ABB RobotStudio station: Aristides_20220202-142745.rsstn

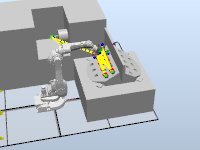
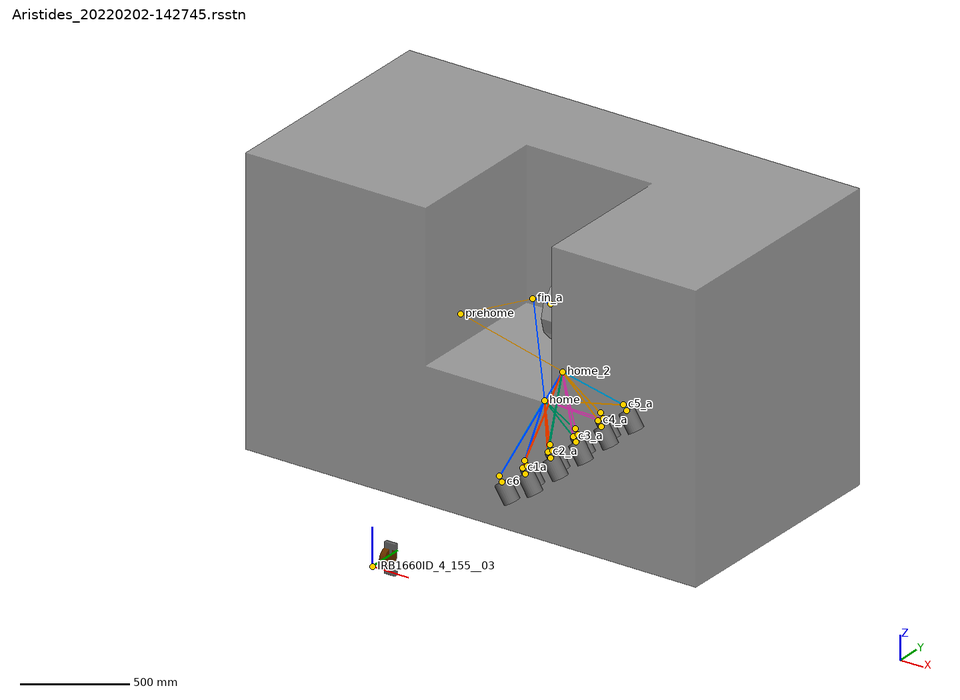
[picture v1: parts stored in the station drawn from their meshes, with robot base, taught points and paths (robot models come from the ABB library and are not in the file)]
Station Aristides (saved by RobotStudio 21.4.9700.0)
Controller Controller3
  mechanical unit ROB_1: IRB1660ID_4_155__03, 6 joints, base frame (0, 0, 0) mm
Layout (positions relative to the parent item):
  - IRB1660ID_4_155__03 [mechanism, from Robots\IRB1660ID_4_155__03.rslib] at (0, 0, 0) mm; joint values [0, 0, 0, 0, 0.5236, 0] (rad or m)
  - Pinza_1 [mechanism, from Efectores_finales - Copy\Pinza_1.rslib] at (944.87, 0, 1229) mm, rotated rx 180 ry 60 rz 180 deg; joint values [0, 0] (rad or m)
  - Torno [part] at (-1172.42, 1966.27, 0) mm, rotated rx 0 ry 0 rz 180 deg, size 2500 x 1300 x 1500 mm
  - Fence_740 [graphiccomponentgroup, from Equipment\Fence_740.rslib] at (-1160.76, -802.49, 0) mm
    - Body 1 [part, from Equipment\Fence_740.rslib]
    - Body 2 [part, from Equipment\Fence_740.rslib]
  - Fence_2500 [graphiccomponentgroup, from Equipment\Fence_2500.rslib] at (1297.15, -826.85, 0) mm, rotated rx 0 ry 0 rz 90 deg
    - Body 1 [part, from Equipment\Fence_2500.rslib]
    - Body 2 [part, from Equipment\Fence_2500.rslib]
  - Fence_740_2 [graphiccomponentgroup, from Equipment\Fence_740.rslib] at (-1148.66, -57.63, 0) mm
    - Body 1 [part, from Equipment\Fence_740.rslib]
    - Body 2 [part, from Equipment\Fence_740.rslib]
  - c5 [part] at (1213.21, 355.81, 885.53) mm, rotated rx 0 ry -32 rz 0 deg, size 80 x 79.4 x 100 mm
  - c3 [part] at (1213.21, -44.2, 885.53) mm, rotated rx 0 ry -32 rz 0 deg, size 80 x 79.4 x 100 mm
  - c2 [part] at (1213.21, -244.19, 885.53) mm, rotated rx 0 ry -32 rz 0 deg, size 80 x 79.4 x 100 mm
  - c8 [part] at (1084.59, -44.2, 808.36) mm, rotated rx 0 ry -32 rz 0 deg, size 80 x 79.4 x 100 mm
  - c4 [part] at (1213.21, 155.81, 885.53) mm, rotated rx 0 ry -32 rz 0 deg, size 80 x 79.4 x 100 mm
  - c7 [part] at (1084.59, -244.19, 808.36) mm, rotated rx 0 ry -32 rz 0 deg, size 80 x 79.4 x 100 mm
  - c6 [part] at (1084.59, -444.19, 808.36) mm, rotated rx 0 ry -32 rz 0 deg, size 80 x 79.4 x 100 mm
  - c9 [part] at (1084.59, 155.81, 808.36) mm, rotated rx 0 ry -32 rz 0 deg, size 80 x 79.4 x 100 mm
  - c10 [part] at (1084.59, 355.81, 808.36) mm, rotated rx 0 ry -32 rz 0 deg, size 80 x 79.4 x 100 mm
  - fin [part] at (377.58, 1016.27, 1000) mm, size 100 x 79.4 x 80 mm
  - c0 [part] at (277.58, 1016.27, 1000) mm, size 100 x 79.4 x 80 mm
  - Positioner [smart component, from Components\Positioner.rslib]
      properties: Object=(none); Position=[0 0 0]; Orientation=[0 0 0]; Reference=Global; ReferenceObject=(none)
  - Detacher [smart component, from Components\Detacher.rslib]
      properties: Child=(none); KeepPosition=true
  - Attacher [smart component, from Components\Attacher.rslib]
      properties: Parent=Pinza_2; Flange=0; Child=(none); Mount=false; Offset=[0 0 0]; Orientation=[0 0 0]
  - CollisionSensor [smart component, from Components\CollisionSensor.rslib]
      properties: Object1=Pinza_2; Object2=c1; NearMiss=0.01; Part1=(none); Part2=(none); CollisionType=0
  - CollisionSensor_2 [smart component, from Components\CollisionSensor.rslib]
      properties: Object1=(none); Object2=(none); NearMiss=0; Part1=(none); Part2=(none); CollisionType=0
  - c1 [part] at (1213.21, -444.19, 885.53) mm, rotated rx 0 ry -32 rz 0 deg, size 80 x 79.4 x 100 mm
  - Efector final 2 [part] at (70, 0, -80) mm, rotated rx 0 ry -90 rz -180 deg, size 100 x 99.5 x 30 mm
  - Pinza1_5 [part] at (130, 10, -10) mm, rotated rx 0 ry 0 rz 180 deg, size 60 x 20 x 60 mm
  - Pinza1_6 [part] at (130, -10, 150) mm, rotated rx 180 ry 0 rz 180 deg, size 60 x 20 x 60 mm
    - Pinza_2_1 [frame] at (30, 10, 80) mm, rotated rx 0 ry -90 rz 0 deg
  - Pinza_2 [mechanism, from Efectores_finales\PINZA2.rslib] at (944.87, 0, 1229) mm, rotated rx 180 ry 60 rz 180 deg; joint values [0, 0] (rad or m)
  - mesa_giratoria [smart component, from Efectores_finales\mesa_giratoria.rslib] at (1381.81, -44.2, 0) mm
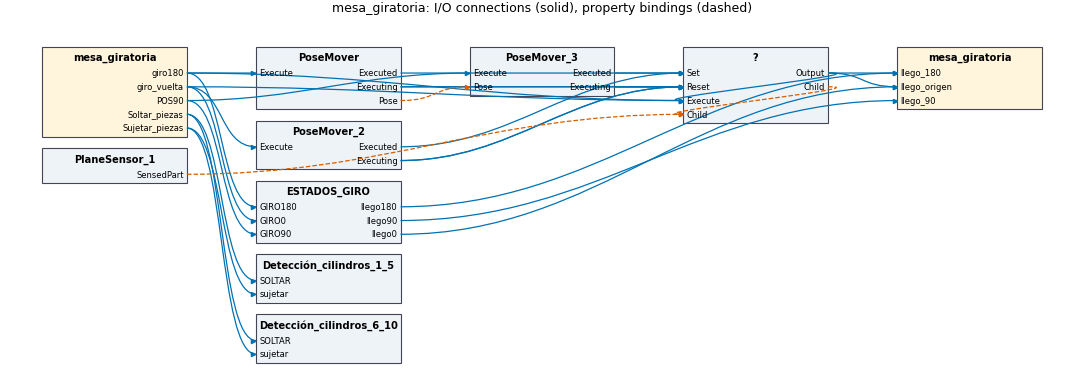
      connections:
        mesa_giratoria.giro180 -> PoseMover.Execute
        mesa_giratoria.giro_vuelta -> PoseMover_2.Execute
        PoseMover.Executed -> ?.Set
        ?.Output -> mesa_giratoria.llego_180
        PoseMover_2.Executed -> ?.Set
        ?.Output -> mesa_giratoria.llego_origen
        PoseMover_2.Executing -> ?.Reset
        PoseMover.Executing -> ?.Reset
        ?.Output -> ?.Execute
        mesa_giratoria.giro_vuelta -> ?.Execute
        mesa_giratoria.giro180 -> ?.Execute
        mesa_giratoria.POS90 -> PoseMover_3.Execute
        PoseMover_3.Executed -> ?.Set
        PoseMover.Executing -> ?.Reset
        PoseMover_2.Executing -> ?.Reset
        PoseMover_3.Executing -> ?.Reset
        PoseMover_3.Executing -> ?.Reset
        mesa_giratoria.giro180 -> ESTADOS_GIRO.GIRO180
        mesa_giratoria.giro_vuelta -> ESTADOS_GIRO.GIRO0
        mesa_giratoria.POS90 -> ESTADOS_GIRO.GIRO90
        ESTADOS_GIRO.llego180 -> mesa_giratoria.llego_180
        ESTADOS_GIRO.llego90 -> mesa_giratoria.llego_90
        ESTADOS_GIRO.llego0 -> mesa_giratoria.llego_origen
        mesa_giratoria.Soltar_piezas -> Detección_cilindros_1_5.SOLTAR
        mesa_giratoria.Soltar_piezas -> Detección_cilindros_6_10.SOLTAR
        mesa_giratoria.Sujetar_piezas -> Detección_cilindros_1_5.sujetar
        mesa_giratoria.Sujetar_piezas -> Detección_cilindros_6_10.sujetar
        PlaneSensor_1.SensedPart => ?.Child
        ?.Child => ?.Child
        PoseMover.Pose => PoseMover_3.Pose
    - Detección_cilindros_6_10 [smart component, from Efectores_finales\mesa_giratoria.rslib]
        connections:
          Detección_cilindros_6_10.SOLTAR -> Deteccion6.liberar
          Detección_cilindros_6_10.SOLTAR -> Deteccion10.liberar
          Detección_cilindros_6_10.SOLTAR -> Deteccion7.liberar
          Detección_cilindros_6_10.SOLTAR -> Deteccion8.liberar
          Detección_cilindros_6_10.SOLTAR -> Deteccion9.liberar
          Detección_cilindros_6_10.sujetar -> Deteccion6.Fijar
          Detección_cilindros_6_10.sujetar -> Deteccion10.Fijar
          Detección_cilindros_6_10.sujetar -> Deteccion7.Fijar
          Detección_cilindros_6_10.sujetar -> Deteccion9.Fijar
          Detección_cilindros_6_10.sujetar -> Deteccion8.Fijar
      - Deteccion6 [smart component, from Efectores_finales\mesa_giratoria.rslib]
        - Attacher_6 [smart component, from Components\Attacher.rslib]
            properties: Parent=Mi_mecanismo; Flange=0; Child=c6; Mount=false; Offset=[0 0 0]; Orientation=[0 0 0]
        - PlaneSensor_6 [smart component, from Components\PlaneSensor.rslib] at (-613.43, 800, 257.08) mm, rotated rx 0 ry 42 rz 0 deg
            properties: Origin=[0.0459897083517545 -0.4 1.14120505334971]; Axis1=[0.0787846202409767 0 0.0138918542133544]; Axis2=[0 0.04 0]; SensedPart=(none)
          - _sensorPart_ [part, from Efectores_finales\mesa_giratoria.rslib]
        - Detacher_6 [smart component, from Components\Detacher.rslib]
            properties: Child=(none); KeepPosition=true
      - Deteccion7 [smart component, from Efectores_finales\mesa_giratoria.rslib]
        - Attacher_7 [smart component, from Components\Attacher.rslib]
            properties: Parent=Mi_mecanismo; Flange=0; Child=c7; Mount=false; Offset=[0 0 0]; Orientation=[0 0 0]
        - PlaneSensor_7 [smart component, from Components\PlaneSensor.rslib] at (-613.43, 600, 257.08) mm, rotated rx 0 ry 42 rz 0 deg
            properties: Origin=[0.0459897083517545 -0.4 1.14120505334971]; Axis1=[0.0787846202409767 0 0.0138918542133544]; Axis2=[0 0.04 0]; SensedPart=(none)
          - _sensorPart_ [part, from Efectores_finales\mesa_giratoria.rslib]
        - Detacher_7 [smart component, from Components\Detacher.rslib]
            properties: Child=(none); KeepPosition=true
      - Deteccion8 [smart component, from Efectores_finales\mesa_giratoria.rslib]
        - Attacher_8 [smart component, from Components\Attacher.rslib]
            properties: Parent=Mi_mecanismo; Flange=0; Child=c8; Mount=false; Offset=[0 0 0]; Orientation=[0 0 0]
        - PlaneSensor_8 [smart component, from Components\PlaneSensor.rslib] at (-613.43, 400, 257.08) mm, rotated rx 0 ry 42 rz 0 deg
            properties: Origin=[0.0459897083517545 -0.4 1.14120505334971]; Axis1=[0.0787846202409767 0 0.0138918542133544]; Axis2=[0 0.04 0]; SensedPart=(none)
          - _sensorPart_ [part, from Efectores_finales\mesa_giratoria.rslib]
        - Detacher_8 [smart component, from Components\Detacher.rslib]
            properties: Child=(none); KeepPosition=true
      - Deteccion9 [smart component, from Efectores_finales\mesa_giratoria.rslib]
        - PlaneSensor_9 [smart component, from Components\PlaneSensor.rslib] at (-613.43, 0, 257.08) mm, rotated rx 0 ry 42 rz 0 deg
            properties: Origin=[0.0459897083517545 -0.4 1.14120505334971]; Axis1=[0.0787846202409767 0 0.0138918542133544]; Axis2=[0 0.04 0]; SensedPart=(none)
          - _sensorPart_ [part, from Efectores_finales\mesa_giratoria.rslib]
        - Attacher_9 [smart component, from Components\Attacher.rslib]
            properties: Parent=Mi_mecanismo; Flange=0; Child=c9; Mount=true; Offset=[0 0 0]; Orientation=[0 0 0]
        - Detacher_9 [smart component, from Components\Detacher.rslib]
            properties: Child=(none); KeepPosition=true
      - Deteccion10 [smart component, from Efectores_finales\mesa_giratoria.rslib]
        - Attacher_10 [smart component, from Components\Attacher.rslib] at (-100, -800, -200) mm
            properties: Parent=Mi_mecanismo; Flange=0; Child=c10; Mount=false; Offset=[0 0 0]; Orientation=[0 0 0]
        - PlaneSensor_10 [smart component, from Components\PlaneSensor.rslib] at (-613.43, 200, 257.08) mm, rotated rx 0 ry 42 rz 0 deg
            properties: Origin=[0.0459897083517545 -0.4 1.14120505334971]; Axis1=[0.0787846202409767 0 0.0138918542133544]; Axis2=[0 0.04 0]; SensedPart=(none)
          - _sensorPart_ [part, from Efectores_finales\mesa_giratoria.rslib]
        - Detacher_10 [smart component, from Components\Detacher.rslib]
            properties: Child=(none); KeepPosition=true
    - Detección_cilindros_1_5 [smart component, from Efectores_finales\mesa_giratoria.rslib]
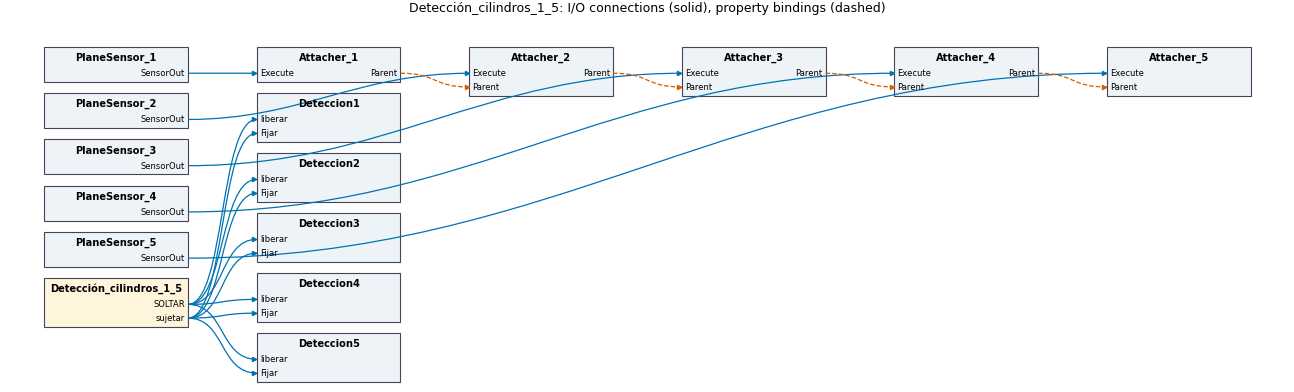
        connections:
          PlaneSensor_1.SensorOut -> Attacher_1.Execute
          PlaneSensor_2.SensorOut -> Attacher_2.Execute
          PlaneSensor_3.SensorOut -> Attacher_3.Execute
          PlaneSensor_4.SensorOut -> Attacher_4.Execute
          PlaneSensor_5.SensorOut -> Attacher_5.Execute
          Detección_cilindros_1_5.SOLTAR -> Deteccion1.liberar
          Detección_cilindros_1_5.sujetar -> Deteccion1.Fijar
          Detección_cilindros_1_5.SOLTAR -> Deteccion2.liberar
          Detección_cilindros_1_5.sujetar -> Deteccion2.Fijar
          Detección_cilindros_1_5.SOLTAR -> Deteccion3.liberar
          Detección_cilindros_1_5.sujetar -> Deteccion3.Fijar
          Detección_cilindros_1_5.SOLTAR -> Deteccion4.liberar
          Detección_cilindros_1_5.sujetar -> Deteccion4.Fijar
          Detección_cilindros_1_5.SOLTAR -> Deteccion5.liberar
          Detección_cilindros_1_5.sujetar -> Deteccion5.Fijar
          Attacher_1.Parent => Attacher_2.Parent
          Attacher_2.Parent => Attacher_3.Parent
          Attacher_3.Parent => Attacher_4.Parent
          Attacher_4.Parent => Attacher_5.Parent
      - Deteccion1 [smart component, from Efectores_finales\mesa_giratoria.rslib]
          connections:
            Deteccion1.liberar -> Detacher_1.Execute
            Deteccion1.Fijar -> Attacher_2.Execute
            Attacher_1.Child => Detacher_1.Child
            PlaneSensor_1.SensedPart => Attacher_2.Child
        - Attacher_1 [smart component, from Components\Attacher.rslib] at (-100, 0, -200) mm
            properties: Parent=Mi_mecanismo; Flange=0; Child=c1; Mount=false; Offset=[0 0 0]; Orientation=[0 0 0]
        - PlaneSensor_1 [smart component, from Components\PlaneSensor.rslib] at (-742.06, 0, 334.25) mm, rotated rx 0 ry 42 rz 0 deg
            properties: Origin=[0.0459897083517545 -0.4 1.14120505334971]; Axis1=[0.0787846202409767 0 0.0138918542133544]; Axis2=[0 0.04 0]; SensedPart=(none)
          - _sensorPart_ [part, from Efectores_finales\mesa_giratoria.rslib]
        - Detacher_1 [smart component, from Components\Detacher.rslib]
            properties: Child=c1; KeepPosition=true
        - Attacher_2 [smart component, from Components\Attacher.rslib]
            properties: Parent=(none); Flange=0; Child=(none); Mount=false; Offset=[0 0 0]; Orientation=[0 0 0]
      - Deteccion2 [smart component, from Efectores_finales\mesa_giratoria.rslib]
          connections:
            Attacher_2.Child => Detacher_2.Child
        - Attacher_2 [smart component, from Components\Attacher.rslib] at (-100, 0, -200) mm
            properties: Parent=Mi_mecanismo; Flange=0; Child=c2; Mount=false; Offset=[0 0 0]; Orientation=[0 0 0]
        - PlaneSensor_2 [smart component, from Components\PlaneSensor.rslib] at (-742.06, 200, 334.25) mm, rotated rx 0 ry 42 rz 0 deg
            properties: Origin=[0.0459897083517545 -0.4 1.14120505334971]; Axis1=[0.0787846202409767 0 0.0138918542133544]; Axis2=[0 0.04 0]; SensedPart=(none)
          - _sensorPart_ [part, from Efectores_finales\mesa_giratoria.rslib]
        - Detacher_2 [smart component, from Components\Detacher.rslib]
            properties: Child=c2; KeepPosition=true
      - Deteccion3 [smart component, from Efectores_finales\mesa_giratoria.rslib]
        - Attacher_3 [smart component, from Components\Attacher.rslib]
            properties: Parent=Mi_mecanismo; Flange=0; Child=c3; Mount=false; Offset=[0 0 0]; Orientation=[0 0 0]
        - PlaneSensor_3 [smart component, from Components\PlaneSensor.rslib] at (-742.06, 400, 334.25) mm, rotated rx 0 ry 42 rz 0 deg
            properties: Origin=[0.0459897083517545 -0.4 1.14120505334971]; Axis1=[0.0787846202409767 0 0.0138918542133544]; Axis2=[0 0.04 0]; SensedPart=(none)
          - _sensorPart_ [part, from Efectores_finales\mesa_giratoria.rslib]
        - Detacher_3 [smart component, from Components\Detacher.rslib]
            properties: Child=(none); KeepPosition=true
      - Deteccion4 [smart component, from Efectores_finales\mesa_giratoria.rslib]
        - Attacher_4 [smart component, from Components\Attacher.rslib]
            properties: Parent=Mi_mecanismo; Flange=0; Child=c4; Mount=false; Offset=[0 0 0]; Orientation=[0 0 0]
        - PlaneSensor_4 [smart component, from Components\PlaneSensor.rslib] at (-742.06, 600, 334.25) mm, rotated rx 0 ry 42 rz 0 deg
            properties: Origin=[0.0459897083517545 -0.4 1.14120505334971]; Axis1=[0.0787846202409767 0 0.0138918542133544]; Axis2=[0 0.04 0]; SensedPart=(none)
          - _sensorPart_ [part, from Efectores_finales\mesa_giratoria.rslib]
        - Detacher_4 [smart component, from Components\Detacher.rslib]
            properties: Child=(none); KeepPosition=true
      - Deteccion5 [smart component, from Efectores_finales\mesa_giratoria.rslib]
        - Attacher_5 [smart component, from Components\Attacher.rslib]
            properties: Parent=Mi_mecanismo; Flange=0; Child=c5; Mount=false; Offset=[0 0 0]; Orientation=[0 0 0]
        - PlaneSensor_5 [smart component, from Components\PlaneSensor.rslib] at (-742.06, 800, 334.25) mm, rotated rx 0 ry 42 rz 0 deg
            properties: Origin=[0.0459897083517545 -0.4 1.14120505334971]; Axis1=[0.0787846202409767 0 0.0138918542133544]; Axis2=[0 0.04 0]; SensedPart=(none)
          - _sensorPart_ [part, from Efectores_finales\mesa_giratoria.rslib]
        - Detacher_5 [smart component, from Components\Detacher.rslib]
            properties: Child=(none); KeepPosition=true
    - c1_1 [part, from Efectores_finales\mesa_giratoria.rslib] at (-31.4, -400, 885.53) mm, rotated rx 0 ry -30 rz 180 deg
    - c2 [part, from Efectores_finales\mesa_giratoria.rslib] at (-168.6, 200, 885.53) mm, rotated rx 0 ry -30 rz 0 deg
    - c2_1 [part, from Efectores_finales\mesa_giratoria.rslib] at (68.6, -200, 1085.53) mm, rotated rx 0 ry -30 rz 180 deg
    - c3 [part, from Efectores_finales\mesa_giratoria.rslib] at (-168.6, 0, 885.53) mm, rotated rx 0 ry -30 rz 0 deg
    - c3_1 [part, from Efectores_finales\mesa_giratoria.rslib] at (68.6, 0, 1085.53) mm, rotated rx 0 ry -30 rz 180 deg
    - c4 [part, from Efectores_finales\mesa_giratoria.rslib] at (-168.6, -200, 885.53) mm, rotated rx 0 ry -30 rz 0 deg
    - c4_1 [part, from Efectores_finales\mesa_giratoria.rslib] at (68.6, 200, 1085.53) mm, rotated rx 0 ry -30 rz 180 deg
    - c5 [part, from Efectores_finales\mesa_giratoria.rslib] at (-168.6, -400, 885.53) mm, rotated rx 0 ry -30 rz 0 deg
    - c5_1 [part, from Efectores_finales\mesa_giratoria.rslib] at (68.6, 400, 1085.53) mm, rotated rx 0 ry -30 rz 180 deg
    - c6 [part, from Efectores_finales\mesa_giratoria.rslib] at (-297.22, -400, 808.36) mm, rotated rx 0 ry -30 rz 0 deg
    - c6_1 [part, from Efectores_finales\mesa_giratoria.rslib] at (197.22, 400, 1008.36) mm, rotated rx 0 ry -30 rz 180 deg
    - c7 [part, from Efectores_finales\mesa_giratoria.rslib] at (-297.22, -200, 808.36) mm, rotated rx 0 ry -30 rz 0 deg
    - c7_1 [part, from Efectores_finales\mesa_giratoria.rslib] at (197.22, 200, 1008.36) mm, rotated rx 0 ry -30 rz 180 deg
    - c8 [part, from Efectores_finales\mesa_giratoria.rslib] at (-297.95, 0, 807.93) mm, rotated rx 0 ry 30 rz 180 deg
    - c8_1 [part, from Efectores_finales\mesa_giratoria.rslib] at (197.95, 0, 1007.93) mm, rotated rx 0 ry 30 rz 0 deg
    - c9 [part, from Efectores_finales\mesa_giratoria.rslib] at (-297.22, 200, 808.36) mm, rotated rx 0 ry 30 rz 180 deg
    - c9_1 [part, from Efectores_finales\mesa_giratoria.rslib] at (197.22, -200, 1008.36) mm, rotated rx 0 ry 30 rz 0 deg
    - c10 [part, from Efectores_finales\mesa_giratoria.rslib] at (-297.22, 400, 808.36) mm, rotated rx 0 ry -30 rz 0 deg
    - c10_1 [part, from Efectores_finales\mesa_giratoria.rslib] at (197.22, -400, 1008.36) mm, rotated rx 0 ry -30 rz 180 deg
    - Mi_mecanismo [mechanism, from Efectores_finales\mesa_giratoria.rslib] at (-100, 0, -200) mm; joint values [0, 0] (rad or m)
    - ESTADOS_GIRO [smart component, from Efectores_finales\mesa_giratoria.rslib]
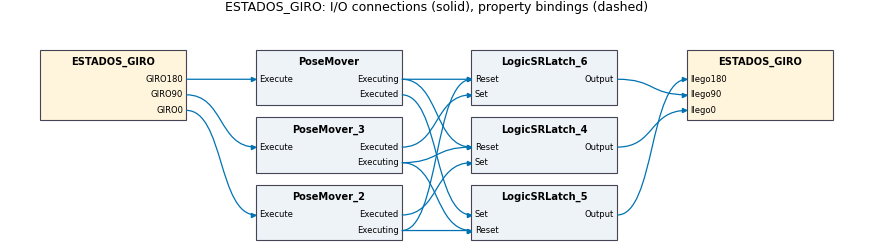
        connections:
          ESTADOS_GIRO.GIRO180 -> PoseMover.Execute
          ESTADOS_GIRO.GIRO90 -> PoseMover_3.Execute
          ESTADOS_GIRO.GIRO0 -> PoseMover_2.Execute
          PoseMover.Executing -> LogicSRLatch_6.Reset
          PoseMover.Executing -> LogicSRLatch_4.Reset
          PoseMover.Executed -> LogicSRLatch_5.Set
          PoseMover_3.Executed -> LogicSRLatch_6.Set
          PoseMover_2.Executed -> LogicSRLatch_4.Set
          PoseMover_3.Executing -> LogicSRLatch_5.Reset
          PoseMover_3.Executing -> LogicSRLatch_4.Reset
          PoseMover_2.Executing -> LogicSRLatch_6.Reset
          PoseMover_2.Executing -> LogicSRLatch_5.Reset
          LogicSRLatch_5.Output -> ESTADOS_GIRO.llego180
          LogicSRLatch_6.Output -> ESTADOS_GIRO.llego90
          LogicSRLatch_4.Output -> ESTADOS_GIRO.llego0
      - PoseMover [smart component, from Components\PoseMover.rslib]
          properties: Mechanism=Mi_mecanismo; Pose=1; Duration=4
      - PoseMover_2 [smart component, from Components\PoseMover.rslib]
          properties: Mechanism=Mi_mecanismo; Pose=2; Duration=4
      - PoseMover_3 [smart component, from Components\PoseMover.rslib]
          properties: Mechanism=Mi_mecanismo; Pose=3; Duration=4
      - LogicSRLatch_4 [smart component, from Components\LogicSRLatch.rslib]
      - LogicSRLatch_5 [smart component, from Components\LogicSRLatch.rslib]
      - LogicSRLatch_6 [smart component, from Components\LogicSRLatch.rslib]
    - c1 [part, from Efectores_finales\mesa_giratoria.rslib] at (-168.6, 400, 885.53) mm, rotated rx 0 ry -30 rz 0 deg
Attachment: Pinza_2 is attached to IRB1660ID_4_155__03 / Link6
Attachment: Pinza_1 is attached to IRB1660ID_4_155__03 / Link6
Attachment: Attacher_10 is attached to c6
Attachment: Attacher_1 is attached to Mi_mecanismo / L3
Attachment: Attacher_2 is attached to Mi_mecanismo / L3
Attachment: c2 is attached to Mi_mecanismo / L3
Attachment: c3 is attached to Mi_mecanismo / L3
Attachment: c4 is attached to Mi_mecanismo / L3
Attachment: c5 is attached to Mi_mecanismo / L3
Attachment: c6 is attached to Mi_mecanismo / L3
Attachment: c7 is attached to Mi_mecanismo / L3
Attachment: c8 is attached to Mi_mecanismo / L3
Attachment: c9 is attached to Mi_mecanismo / L3
Attachment: c10 is attached to Mi_mecanismo / L3
Attachment: c1 is attached to Mi_mecanismo / L3
Station logic (signal -> signal, property => property):
  CollisionSensor.SensorOut -> Attacher.Execute
  CollisionSensor.Object1 => Attacher.Parent
  CollisionSensor.Part2 => Attacher.Child
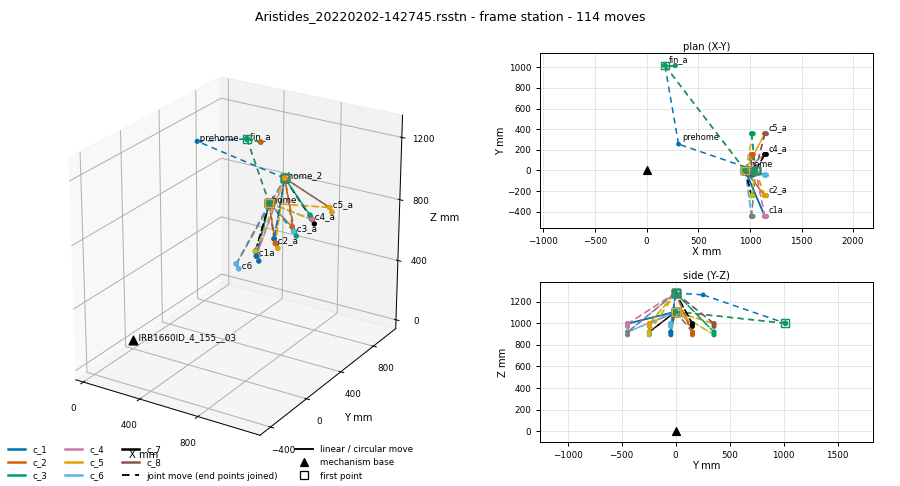
[picture p0: tool path of Aristides_20220202-142745.rsstn in frame station, 114 of 114 moves have a stored position in this frame; points joined in program order, loops and branches not executed]
Targets, tools, work objects and paths stored in the station, written as RAPID:
! task T_ROB1
MODULE Module1
  CONST robtarget home:=[[955.495207776,0,1107.397459622],[0.258819045,0,-0.965925826,0],[0,0,0,0],[9E+09,9E+09,9E+09,9E+09,9E+09,9E+09]];
  CONST robtarget c1:=[[1160.221,-444.195,970.335],[0.275637356,0,0.961261696,0],[-1,1,-2,0],[9E+09,9E+09,9E+09,9E+09,9E+09,9E+09]];
  CONST robtarget c1a:=[[1144.323422065,-444.195,995.77644288],[0.275637356,0,0.961261696,0],[-1,1,-2,0],[9E+09,9E+09,9E+09,9E+09,9E+09,9E+09]];
  CONST robtarget c2:=[[1160.221,-244.195,970.335],[0.275637356,0,0.961261696,0],[-1,1,-2,0],[9E+09,9E+09,9E+09,9E+09,9E+09,9E+09]];
  CONST robtarget c2_a:=[[1144.323422065,-244.195,995.77644288],[0.275637356,0,0.961261696,0],[-1,1,-2,0],[9E+09,9E+09,9E+09,9E+09,9E+09,9E+09]];
  CONST robtarget c3:=[[1160.221,-44.195,970.335],[0.275637356,0,0.961261696,0],[-1,-1,0,1],[9E+09,9E+09,9E+09,9E+09,9E+09,9E+09]];
  CONST robtarget c3_a:=[[1144.323422065,-44.195,995.77644288],[0.275637356,0,0.961261696,0],[-1,-1,0,1],[9E+09,9E+09,9E+09,9E+09,9E+09,9E+09]];
  CONST robtarget c4:=[[1160.221,155.805,970.335],[0.275637356,0,0.961261696,0],[0,-2,1,0],[9E+09,9E+09,9E+09,9E+09,9E+09,9E+09]];
  CONST robtarget c4_a:=[[1144.323422065,155.805,995.77644288],[0.275637356,0,0.961261696,0],[0,-2,1,0],[9E+09,9E+09,9E+09,9E+09,9E+09,9E+09]];
  CONST robtarget c5:=[[1160.221,355.805,970.335],[0.275637356,0,0.961261696,0],[0,-2,1,0],[9E+09,9E+09,9E+09,9E+09,9E+09,9E+09]];
  CONST robtarget c5_a:=[[1144.323422065,355.805,995.77644288],[0.275637356,0,0.961261696,0],[0,-2,1,0],[9E+09,9E+09,9E+09,9E+09,9E+09,9E+09]];
  CONST robtarget c6:=[[1031.597,-444.195,893.161],[0.275637356,0,0.961261696,0],[-1,1,-2,0],[9E+09,9E+09,9E+09,9E+09,9E+09,9E+09]];
  CONST robtarget c6_a:=[[1015.699422065,-444.195,918.60244288],[0.275637356,0,0.961261696,0],[-1,1,-2,0],[9E+09,9E+09,9E+09,9E+09,9E+09,9E+09]];
  CONST robtarget c7:=[[1031.597,-244.195,893.161],[0.275637356,0,0.961261696,0],[-1,1,-2,0],[9E+09,9E+09,9E+09,9E+09,9E+09,9E+09]];
  CONST robtarget c7_a:=[[1015.699422065,-244.195,918.60244288],[0.275637356,0,0.961261696,0],[-1,1,-2,0],[9E+09,9E+09,9E+09,9E+09,9E+09,9E+09]];
  CONST robtarget c8:=[[1031.597,-44.195,893.161],[0.275637356,0,0.961261696,0],[-1,-1,0,1],[9E+09,9E+09,9E+09,9E+09,9E+09,9E+09]];
  CONST robtarget c8_a:=[[1015.699422065,-44.195,918.60244288],[0.275637356,0,0.961261696,0],[-1,-1,0,1],[9E+09,9E+09,9E+09,9E+09,9E+09,9E+09]];
  CONST robtarget c9_a:=[[1015.699422065,155.805,918.60244288],[0.275637356,0,0.961261696,0],[0,-2,1,0],[9E+09,9E+09,9E+09,9E+09,9E+09,9E+09]];
  CONST robtarget c9:=[[1031.597,155.805,893.161],[0.275637356,0,0.961261696,0],[0,-2,1,0],[9E+09,9E+09,9E+09,9E+09,9E+09,9E+09]];
  CONST robtarget c10:=[[1031.597,355.805,893.161],[0.275637356,0,0.961261696,0],[0,-2,1,0],[9E+09,9E+09,9E+09,9E+09,9E+09,9E+09]];
  CONST robtarget c10_a:=[[1031.597,355.805,893.161],[0.275637356,0,0.961261696,0],[0,-2,1,0],[9E+09,9E+09,9E+09,9E+09,9E+09,9E+09]];
  CONST robtarget fin_a:=[[177.584,1016.268,1000],[0.5,0.5,0.5,0.5],[0,1,-1,0],[9E+09,9E+09,9E+09,9E+09,9E+09,9E+09]];
  CONST robtarget fin:=[[277.584,1016.268,1000],[0.5,0.5,0.5,0.5],[0,1,-1,0],[9E+09,9E+09,9E+09,9E+09,9E+09,9E+09]];
  CONST robtarget home_2:=[[1055.495207776,0,1280.602540378],[0.965925826,0,0.258819045,0],[0,0,0,0],[9E+09,9E+09,9E+09,9E+09,9E+09,9E+09]];
  CONST robtarget final_a:=[[177.584,1016.268,1000],[0.5,-0.5,0.5,-0.5],[0,0,0,0],[9E+09,9E+09,9E+09,9E+09,9E+09,9E+09]];
  CONST robtarget final:=[[277.584,1016.268,1000],[0.5,-0.5,0.5,-0.5],[0,1,1,0],[9E+09,9E+09,9E+09,9E+09,9E+09,9E+09]];
  CONST robtarget prehome:=[[309.604,254.998,1262.538],[0.396697298,0.585347123,0.410036045,0.576081975],[0,1,0,0],[9E+09,9E+09,9E+09,9E+09,9E+09,9E+09]];
  CONST robtarget c1_3:=[[1160.221,-444.195,970.335],[0,0.961261696,0,0.275637356],[-1,1,0,0],[9E+09,9E+09,9E+09,9E+09,9E+09,9E+09]];
  CONST robtarget c1a_3:=[[1144.323422065,-444.195,995.77644288],[0,0.961261696,0,0.275637356],[-1,1,0,0],[9E+09,9E+09,9E+09,9E+09,9E+09,9E+09]];
  CONST robtarget c2_3:=[[1160.221,-244.195,970.335],[0,0.961261696,0,0.275637356],[-1,1,0,0],[9E+09,9E+09,9E+09,9E+09,9E+09,9E+09]];
  CONST robtarget c2_a_2:=[[1144.323422065,-244.195,995.77644288],[0,0.961261696,0,0.275637356],[-1,1,0,0],[9E+09,9E+09,9E+09,9E+09,9E+09,9E+09]];
  CONST robtarget c3_3:=[[1160.221,-44.195,970.335],[0,0.961261696,0,0.275637356],[-1,-1,-2,1],[9E+09,9E+09,9E+09,9E+09,9E+09,9E+09]];
  CONST robtarget c3_a_2:=[[1144.323422065,-44.195,995.77644288],[0,0.961261696,0,0.275637356],[-1,-1,-2,1],[9E+09,9E+09,9E+09,9E+09,9E+09,9E+09]];
  CONST robtarget c4_3:=[[1160.221,155.805,970.335],[0,0.961261696,0,0.275637356],[0,-2,-1,0],[9E+09,9E+09,9E+09,9E+09,9E+09,9E+09]];
  CONST robtarget c4_a_2:=[[1144.323422065,155.805,995.77644288],[0,0.961261696,0,0.275637356],[0,-2,-1,0],[9E+09,9E+09,9E+09,9E+09,9E+09,9E+09]];
  CONST robtarget c5_3:=[[1160.221,355.805,970.335],[0,0.961261696,0,0.275637356],[0,-2,-1,0],[9E+09,9E+09,9E+09,9E+09,9E+09,9E+09]];
  CONST robtarget c5_a_2:=[[1144.323422065,355.805,995.77644288],[0,0.961261696,0,0.275637356],[0,-2,-1,0],[9E+09,9E+09,9E+09,9E+09,9E+09,9E+09]];
  CONST robtarget c6_3:=[[1031.597,-444.195,893.161],[0,0.961261696,0,0.275637356],[-1,1,0,0],[9E+09,9E+09,9E+09,9E+09,9E+09,9E+09]];
  CONST robtarget c6_a_2:=[[1015.699422065,-444.195,918.60244288],[0,0.961261696,0,0.275637356],[-1,1,0,0],[9E+09,9E+09,9E+09,9E+09,9E+09,9E+09]];
  CONST robtarget c7_3:=[[1031.597,-244.195,893.161],[0,0.961261696,0,0.275637356],[-1,1,0,0],[9E+09,9E+09,9E+09,9E+09,9E+09,9E+09]];
  CONST robtarget c7_a_2:=[[1015.699422065,-244.195,918.60244288],[0,0.961261696,0,0.275637356],[-1,1,0,0],[9E+09,9E+09,9E+09,9E+09,9E+09,9E+09]];
  CONST robtarget c8_3:=[[1031.597,-44.195,893.161],[0,0.961261696,0,0.275637356],[-1,-1,-2,1],[9E+09,9E+09,9E+09,9E+09,9E+09,9E+09]];
  CONST robtarget c8_a_2:=[[1015.699422065,-44.195,918.60244288],[0,0.961261696,0,0.275637356],[-1,-1,-2,1],[9E+09,9E+09,9E+09,9E+09,9E+09,9E+09]];
  CONST robtarget c9_2:=[[1031.597,155.805,893.161],[0,0.961261696,0,0.275637356],[0,-2,-1,0],[9E+09,9E+09,9E+09,9E+09,9E+09,9E+09]];
  CONST robtarget c9_a_3:=[[1015.699422065,155.805,918.60244288],[0,0.961261696,0,0.275637356],[0,-2,-1,0],[9E+09,9E+09,9E+09,9E+09,9E+09,9E+09]];
  CONST robtarget c10_3:=[[1031.597,355.805,893.161],[0,0.961261696,0,0.275637356],[0,-2,-1,0],[9E+09,9E+09,9E+09,9E+09,9E+09,9E+09]];
  CONST robtarget c10_a_2:=[[1015.699422065,355.805,918.60244288],[0,0.961261696,0,0.275637356],[0,-2,-1,0],[9E+09,9E+09,9E+09,9E+09,9E+09,9E+09]];
  PROC main()
    c_1;
    c_1_2;
    c_2;
    c_2_2;
    c_3;
    c_3_2;
    c_4;
    c_4_2;
    c_5;
    c_5_2;
    c_6;
    c_6_2;
    c_7;
    c_7_2;
    c_8;
    c_8_2;
    c_9;
    c_10;
    c_9_2;
    c_10_2;
    giro;
    torno;
  ENDPROC
  PROC c_1()
    MoveJ home,v1000,z100,Pinza_2_1\WObj:=Workobject_2;
    MoveL c1a,v1000,z100,Pinza_2_1\WObj:=Workobject_2;
    MoveL c1,v1000,fine,Pinza_2_1\WObj:=Workobject_2;
    MoveL c1a,v1000,z100,Pinza_2_1\WObj:=Workobject_2;
    MoveL home,v1000,z100,Pinza_2_1\WObj:=Workobject_2;
  ENDPROC
  PROC c_2()
    MoveJ home,v1000,z100,Pinza_2_1\WObj:=Workobject_2;
    MoveJ c2_a,v1000,z100,Pinza_2_1\WObj:=Workobject_2;
    MoveJ c2,v1000,z100,Pinza_2_1\WObj:=Workobject_2;
    MoveJ c2_a,v1000,z100,Pinza_2_1\WObj:=Workobject_2;
    MoveJ home,v1000,z100,Pinza_2_1\WObj:=Workobject_2;
  ENDPROC
  PROC c_3()
    MoveJ home,v1000,z100,Pinza_2_1\WObj:=Workobject_2;
    MoveJ c3_a,v1000,z100,Pinza_2_1\WObj:=Workobject_2;
    MoveJ c3,v1000,z100,Pinza_2_1\WObj:=Workobject_2;
    MoveJ c3_a,v1000,z100,Pinza_2_1\WObj:=Workobject_2;
    MoveJ home,v1000,z100,Pinza_2_1\WObj:=Workobject_2;
  ENDPROC
  PROC c_4()
    MoveJ home,v1000,z100,Pinza_2_1\WObj:=Workobject_2;
    MoveJ c4_a,v1000,z100,Pinza_2_1\WObj:=Workobject_2;
    MoveJ c4,v1000,z100,Pinza_2_1\WObj:=Workobject_2;
    MoveJ c4_a,v1000,z100,Pinza_2_1\WObj:=Workobject_2;
    MoveJ home,v1000,z100,Pinza_2_1\WObj:=Workobject_2;
  ENDPROC
  PROC c_5()
    MoveJ home,v1000,z100,Pinza_2_1\WObj:=Workobject_2;
    MoveJ c5_a,v1000,z100,Pinza_2_1\WObj:=Workobject_2;
    MoveJ c5,v1000,z100,Pinza_2_1\WObj:=Workobject_2;
    MoveJ c5_a,v1000,z100,Pinza_2_1\WObj:=Workobject_2;
    MoveJ home,v1000,z100,Pinza_2_1\WObj:=Workobject_2;
  ENDPROC
  PROC c_6()
    MoveJ home,v1000,z100,Pinza_2_1\WObj:=Workobject_2;
    MoveJ c6_a,v1000,z100,Pinza_2_1\WObj:=Workobject_2;
    MoveJ c6,v1000,z100,Pinza_2_1\WObj:=Workobject_2;
    MoveJ c6_a,v1000,z100,Pinza_2_1\WObj:=Workobject_2;
    MoveJ home,v1000,z100,Pinza_2_1\WObj:=Workobject_2;
  ENDPROC
  PROC c_7()
    MoveJ home,v1000,z100,Pinza_2_1\WObj:=Workobject_2;
    MoveJ c7_a,v1000,z100,Pinza_2_1\WObj:=Workobject_2;
    MoveJ c7,v1000,z100,Pinza_2_1\WObj:=Workobject_2;
    MoveJ c7_a,v1000,z100,Pinza_2_1\WObj:=Workobject_2;
    MoveJ home,v1000,z100,Pinza_2_1\WObj:=Workobject_2;
  ENDPROC
  PROC c_8()
    MoveJ home,v1000,z100,Pinza_2_1\WObj:=Workobject_2;
    MoveJ c8_a,v1000,z100,Pinza_2_1\WObj:=Workobject_2;
    MoveJ c8,v1000,z100,Pinza_2_1\WObj:=Workobject_2;
    MoveJ c8_a,v1000,z100,Pinza_2_1\WObj:=Workobject_2;
    MoveJ home,v1000,z100,Pinza_2_1\WObj:=Workobject_2;
  ENDPROC
  PROC c_9()
    MoveJ home,v1000,z100,Pinza_2_1\WObj:=Workobject_2;
    MoveJ c9_a,v1000,z100,Pinza_2_1\WObj:=Workobject_2;
    MoveJ c9,v1000,z100,Pinza_2_1\WObj:=Workobject_2;
    MoveJ c9_a,v1000,z100,Pinza_2_1\WObj:=Workobject_2;
    MoveJ home,v1000,z100,Pinza_2_1\WObj:=Workobject_2;
  ENDPROC
  PROC c_10()
    MoveJ home,v1000,z100,Pinza_2_1\WObj:=Workobject_2;
    MoveJ c10_a,v1000,z100,Pinza_2_1\WObj:=Workobject_2;
    MoveJ c10,v1000,z100,Pinza_2_1\WObj:=Workobject_2;
    MoveJ c10_a,v1000,z100,Pinza_2_1\WObj:=Workobject_2;
    MoveJ home,v1000,z100,Pinza_2_1\WObj:=Workobject_2;
  ENDPROC
  PROC torno()
    MoveJ home_2,v1000,z100,Pinza_1\WObj:=Workobject_4;
    MoveJ prehome,v1000,z100,Pinza_1\WObj:=Workobject_4;
    MoveJ fin_a,v1000,z100,Pinza_1\WObj:=Workobject_4;
    MoveJ fin,v1000,z100,Pinza_1\WObj:=Workobject_4;
    MoveJ fin_a,v1000,z100,Pinza_1\WObj:=Workobject_4;
  ENDPROC
  PROC giro()
    MoveJ final_a,v1000,z100,tool0\WObj:=Workobject_2;
    MoveJ final,v1000,z100,tool0\WObj:=Workobject_2;
    MoveJ final_a,v1000,z100,tool0\WObj:=Workobject_2;
    MoveJ home,v1000,z100,tool0\WObj:=Workobject_2;
  ENDPROC
  PROC Path_10()
    MoveJ final_a,v1000,z100,tool0\WObj:=Workobject_2;
    MoveJ final,v1000,z100,tool0\WObj:=Workobject_2;
    MoveJ final_a,v1000,z100,tool0\WObj:=Workobject_2;
    MoveJ home,v1000,z100,tool0\WObj:=Workobject_2;
  ENDPROC
  PROC c_1_2()
    MoveJ home_2,v1000,z100,Pinza_1\WObj:=Workobject_4;
    MoveJ c1a_3,v1000,z100,Pinza_1\WObj:=Workobject_4;
    MoveJ c1_3,v1000,z100,Pinza_1\WObj:=Workobject_4;
    MoveJ c1a_3,v1000,z100,Pinza_1\WObj:=Workobject_4;
    MoveJ home_2,v1000,z100,Pinza_1\WObj:=Workobject_4;
  ENDPROC
  PROC c_2_2()
    MoveJ home_2,v1000,z100,Pinza_1\WObj:=Workobject_4;
    MoveJ c2_a_2,v1000,z100,Pinza_1\WObj:=Workobject_4;
    MoveJ c2_3,v1000,z100,Pinza_1\WObj:=Workobject_4;
    MoveJ c2_a_2,v1000,z100,Pinza_1\WObj:=Workobject_4;
    MoveJ home_2,v1000,z100,Pinza_1\WObj:=Workobject_4;
  ENDPROC
  PROC c_3_2()
    MoveJ home_2,v1000,z100,Pinza_1\WObj:=Workobject_4;
    MoveJ c3_a_2,v1000,z100,Pinza_1\WObj:=Workobject_4;
    MoveJ c3_3,v1000,z100,Pinza_1\WObj:=Workobject_4;
    MoveJ c3_a_2,v1000,z100,Pinza_1\WObj:=Workobject_4;
    MoveJ home_2,v1000,z100,Pinza_1\WObj:=Workobject_4;
  ENDPROC
  PROC c_4_2()
    MoveJ home_2,v1000,z100,Pinza_1\WObj:=Workobject_4;
    MoveJ c4_a_2,v1000,z100,Pinza_1\WObj:=Workobject_4;
    MoveJ c4_3,v1000,z100,Pinza_1\WObj:=Workobject_4;
    MoveJ c4_a_2,v1000,z100,Pinza_1\WObj:=Workobject_4;
    MoveJ home_2,v1000,z100,Pinza_1\WObj:=Workobject_4;
  ENDPROC
  PROC c_5_2()
    MoveJ home_2,v1000,z100,Pinza_1\WObj:=Workobject_4;
    MoveJ c5_a_2,v1000,z100,Pinza_1\WObj:=Workobject_4;
    MoveJ c5_3,v1000,z100,Pinza_1\WObj:=Workobject_4;
    MoveJ c5_a_2,v1000,z100,Pinza_1\WObj:=Workobject_4;
    MoveJ home_2,v1000,z100,Pinza_1\WObj:=Workobject_4;
  ENDPROC
  PROC c_6_2()
    MoveJ home_2,v1000,z100,Pinza_1\WObj:=Workobject_4;
    MoveJ c6_a_2,v1000,z100,Pinza_1\WObj:=Workobject_4;
    MoveJ c6_3,v1000,z100,Pinza_1\WObj:=Workobject_4;
    MoveJ c6_a_2,v1000,z100,Pinza_1\WObj:=Workobject_4;
    MoveJ home_2,v1000,z100,Pinza_1\WObj:=Workobject_4;
  ENDPROC
  PROC c_7_2()
    MoveJ home_2,v1000,z100,Pinza_1\WObj:=Workobject_4;
    MoveJ c7_a_2,v1000,z100,Pinza_1\WObj:=Workobject_4;
    MoveJ c7_3,v1000,z100,Pinza_1\WObj:=Workobject_4;
    MoveJ c7_a_2,v1000,z100,Pinza_1\WObj:=Workobject_4;
    MoveJ home_2,v1000,z100,Pinza_1\WObj:=Workobject_4;
  ENDPROC
  PROC c_8_2()
    MoveJ home_2,v1000,z100,Pinza_1\WObj:=Workobject_4;
    MoveJ c8_a_2,v1000,z100,Pinza_1\WObj:=Workobject_4;
    MoveJ c8_3,v1000,z100,Pinza_1\WObj:=Workobject_4;
    MoveJ c8_a_2,v1000,z100,Pinza_1\WObj:=Workobject_4;
    MoveJ home_2,v1000,z100,Pinza_1\WObj:=Workobject_4;
  ENDPROC
  PROC c_9_2()
    MoveJ home_2,v1000,z100,Pinza_1\WObj:=Workobject_4;
    MoveJ c9_a_3,v1000,z100,Pinza_1\WObj:=Workobject_4;
    MoveJ c9_2,v1000,z100,Pinza_1\WObj:=Workobject_4;
    MoveJ c9_a_3,v1000,z100,Pinza_1\WObj:=Workobject_4;
    MoveJ c9_2,v1000,z100,Pinza_1\WObj:=Workobject_4;
    MoveJ home_2,v1000,z100,Pinza_1\WObj:=Workobject_4;
  ENDPROC
  PROC c_10_2()
    MoveJ home_2,v1000,z100,Pinza_1\WObj:=Workobject_4;
    MoveJ c10_a_2,v1000,z100,Pinza_1\WObj:=Workobject_4;
    MoveJ c10_3,v1000,z100,Pinza_1\WObj:=Workobject_4;
    MoveJ c10_a_2,v1000,z100,Pinza_1\WObj:=Workobject_4;
    MoveJ home_2,v1000,z100,Pinza_1\WObj:=Workobject_4;
  ENDPROC
ENDMODULE

! task T_ROB1
MODULE CalibData
  TASK PERS wobjdata Workobject_2:=[FALSE,TRUE,"",[[0,0,0],[1,0,0,0]],[[0,0,0],[1,0,0,0]]];
  TASK PERS wobjdata Workobject_4:=[FALSE,TRUE,"",[[0,0,0],[1,0,0,0]],[[0,0,0],[1,0,0,0]]];
  PERS tooldata Pinza_2_1:=[TRUE,[[140,0,70],[0.707106781,0,0.707106781,0]],[1,[0,0,1],[1,0,0,0],0,0,0]];
  PERS tooldata Pinza_1:=[TRUE,[[-100,0,70],[0.707106781,0,-0.707106781,0]],[1,[0,0,1],[1,0,0,0],0,0,0]];
  PERS tooldata Vara:=[TRUE,[[0,0,250],[0.707106781,0,0,0.707106781]],[1,[0,0,1],[1,0,0,0],0,0,0]];
  PERS tooldata Soplador:=[TRUE,[[0,-70,70],[0.5,0.5,-0.5,0.5]],[1,[0,0,1],[1,0,0,0],0,0,0]];
ENDMODULE

